// TIA Portal V21 export
DATA_BLOCK "Popup"   // DB19
{ S7_Optimized_Access := 'TRUE' }
// stored: MemoryReserve 100
   VAR RETAIN
      P : Array[0.."K_NumPopup"] of "Std_Popup";
   END_VAR
   VAR
      Hmi : Struct
         TriggerPopup : Bool := FALSE;
         IndicePopup : Int := 0;
         ReshowPopUps : Bool := FALSE;
      END_STRUCT;
      Dati : Struct
         NumeroPopUpNonConfermati : Int := 0;
         NumeroPopUpNonConfermatiMemo : Int := 0;
         NumeroPopupConfermati_Nack : Int := 0;
         NumeroPopupConfermati_NackMemo : Int := 0;
      END_STRUCT;
      TimeOutTrigger : "Std_stTimer";
   END_VAR
BEGIN
   P[0..1].RichiestaAperturaPopup := FALSE;
   P[0..1].RichiestaAperturaPopup_Memo := FALSE;
   P[0..1].PopupDaConfermare := FALSE;
   P[0..1].AckOperatore_Inviato := FALSE;
   P[0..1].AckOperatore_Ricevuto := FALSE;
   P[0..1].NackOperatore_Inviato := FALSE;
   P[0..1].NackOperatore_Ricevuto := FALSE;
   P[0..1].ENO_Blocco := FALSE;
   TimeOutTrigger.IN := FALSE;
   TimeOutTrigger.O := FALSE;
   TimeOutTrigger.Preset := 0.6;
   TimeOutTrigger.TempoTrascorso := 0.0;
END_DATA_BLOCK
